(* IEC 61131-3 sources: repolevel_ST_code_completion/output/0121完整版本/repoeval_VisuElements/readful_result_no_provide, 3 files *)

(* ---- MouseEventHandler.st ---- *)
VAR
    LeftClickTimer : TON;
    xLeftClickOld : BOOL;
    iClickCount : INT := 0;
    xEventProcessed : BOOL := FALSE;
    xRightClickOld : BOOL;
    xMiddleClickOld : BOOL;
    xMouseMoveOld : BOOL;
END_VAR

(* Reset event state *)
eMouseEvent := 0;
xEventActive := FALSE;

(* Handle left click events (single/double click) *)
IF xLeftClick AND NOT xLeftClickOld THEN
    IF iClickCount = 0 THEN
        LeftClickTimer(IN := TRUE, PT := tDblClickTime);
        iClickCount := 1;
    ELSE
        LeftClickTimer(IN := FALSE);
        eMouseEvent := 2; (* Double click *)
        rEventX := rMouseX;
        rEventY := rMouseY;
        xEventActive := TRUE;
        iClickCount := 0;
        xEventProcessed := TRUE;
    END_IF
ELSIF NOT xLeftClick AND xLeftClickOld THEN
    IF iClickCount = 1 AND NOT xEventProcessed THEN
        LeftClickTimer();
        IF NOT LeftClickTimer.Q THEN
            (* Waiting for potential double click *)
        END_IF
    END_IF
END_IF

IF LeftClickTimer.Q AND iClickCount = 1 THEN
    eMouseEvent := 1; (* Single click *)
    rEventX := rMouseX;
    rEventY := rMouseY;
    xEventActive := TRUE;
    iClickCount := 0;
END_IF

(* Handle right click events *)
IF xRightClick AND NOT xRightClickOld THEN
    eMouseEvent := 3; (* Right click *)
    rEventX := rMouseX;
    rEventY := rMouseY;
    xEventActive := TRUE;
END_IF

(* Handle middle click events *)
IF xMiddleClick AND NOT xMiddleClickOld THEN
    eMouseEvent := 4; (* Middle click *)
    rEventX := rMouseX;
    rEventY := rMouseY;
    xEventActive := TRUE;
END_IF

(* Handle mouse movement events *)
IF xMouseMove AND NOT xMouseMoveOld THEN
    eMouseEvent := 0; (* Mouse movement does not trigger an event type *)
    rEventX := rMouseX;
    rEventY := rMouseY;
    xEventActive := TRUE;
END_IF

(* Update old states *)
xLeftClickOld := xLeftClick;
xRightClickOld := xRightClick;
xMiddleClickOld := xMiddleClick;
xMouseMoveOld := xMouseMove;
END_FUNCTION_BLOCK

(* ---- NodeExpandCollapse.st ---- *)
VAR
    NodeDblClick : TON;
    xNodeClickOld : BOOL;
    iNodeState : INT := 1;
END_VAR

CASE iNodeState OF
    1: (* Wait for first click *)
        IF xNodeClick AND NOT xNodeClickOld THEN
            NodeDblClick(IN := TRUE, PT := tDblClickTime);
            iNodeState := 2;
            xNodeSelected := TRUE;
        END_IF

    2: (* Wait for second click or timeout *)
        NodeDblClick();
        IF NodeDblClick.Q THEN
            (* Timeout - single click, reset *)
            NodeDblClick(IN := FALSE);
            xNodeClickOld := FALSE;
            iNodeState := 1;
            xNodeSelected := FALSE;
        ELSIF NOT xNodeClick AND xNodeClickOld THEN
            (* Second click detected - toggle expansion *)
            NodeDblClick(IN := FALSE);
            xNodeExpand := NOT xNodeExpand;
            iNodeState := 1;
            xNodeSelected := FALSE;
        END_IF
END_CASE

xNodeClickOld := xNodeClick;
END_FUNCTION_BLOCK

(* ---- RotationCalculation.st ---- *)
VAR
    rRadians : REAL;
    rCos : REAL;
    rSin : REAL;
    rTranslatedX : REAL;
    rTranslatedY : REAL;
END_VAR

rRadians := rAngle * 3.14159265359 / 180.0; // Replace undefined PI with its numeric approximation
rCos := COS(rRadians);          (* Calculate cosine of the angle *)
rSin := SIN(rRadians);          (* Calculate sine of the angle *)

(* Translate point to origin relative to the rotation center *)
rTranslatedX := rPointX - rCenterX;
rTranslatedY := rPointY - rCenterY;

(* Perform rotation *)
rRotatedX := rTranslatedX * rCos - rTranslatedY * rSin + rCenterX;
rRotatedY := rTranslatedX * rSin + rTranslatedY * rCos + rCenterY;

RotationCalculation := TRUE; // Assign result to function name before returning
RETURN; // Exit the function
END_FUNCTION
